FUNCTION_BLOCK icecream_factory
  (* Standard: 61499-2 *)
  (* Version 0,1, 2015-00-16, Th?o, PC_THEO *)
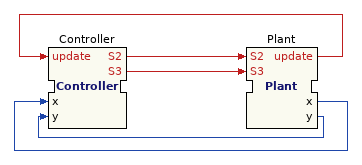
  FBS
    Controller : Controller;
    Plant : Plant;
  END_FBS
  EVENT_CONNECTIONS
    Controller.S2 TO Plant.S2;
    Controller.S3 TO Plant.S3;
    Plant.update TO Controller.update;
  END_CONNECTIONS
  DATA_CONNECTIONS
    Plant.x TO Controller.x;
    Plant.y TO Controller.y;
  END_CONNECTIONS
END_FUNCTION_BLOCK
